TYPE ST_DAR_6_0 :
(**************************************************************************************
 * 	Application		:	BoxControl Framework
 *	Revision		:	$Revision: 404529 $
 *	Revision date	:	$Date: 2018-04-23 08:21:38 +0200 (Mo., 23 Apr 2018) $
 *	Last changed by	:	$Author: b7bolm $
 *	URL				:	$URL: http://almscdc.swisslog.com/repo/SWPD/Development/BoxControlFramework/20_Release/trunk/01_Software/BCF/BCF/JumpStart/20_Product/10_App/11_Com/10_Lib/10_Conv/12_MFCS/11_SIS/01_DUTs/10_SIS_6_0/ST_DAR_6_0.TcDUT $
 *
 *	Purpose			:	DAQ Structure
 *
 * ------------------------------------------------------------------------------------
 *	Copyright Swisslog [IP AG], Switzerland. All rights reserved.
 * 
 * ------------------------------------------------------------------------------------
 *	
 * 	Revision History: 
 *
 * 	VERSION			DATE			INITIALS			DESCRIPTION
 *	0.1				01.01.2001		swl					Example
 *	0.2			    01.01.2016		Sna				    First version
 **************************************************************************************)
STRUCT
	Position 		: STRING(SIS_6_0.POSITION_STRINGLENGTH); // 12 Digit SIS Location MM-GGG-EEEE-FF-Z
	Code			: STRING(SIS_6_0.DATA_ACQUISITION_CODE); // 1 Digit dimension
	NumberOfSets	: STRING(SIS_6_0.DIMENSIONS); // 2 Digit dimension
	Set				: ARRAY[E_CM_Index.E_BEGIN_VARIABLE+1..E_CM_Index.E_END_VARIABLE-1] OF STRING(SIS_6_0.DATA_ACQUISITION_SET); //  maxnumberSets
END_STRUCT
END_TYPE

(* stored: Version 1.1.0.1, ProductVersion 3.1.4022.12
   DUT ST_DAR_6_0: Id {56ae3316-5ca2-477f-aaa0-df69db91e1b1} *)
